INTERFACE I_Logger EXTENDS I_Object

METHOD PUBLIC M_Log
VAR_INPUT
	{attribute 'analysis' := '-33'}
	stEvent	: ST_Event;
END_VAR
END_METHOD

METHOD PUBLIC M_Reset
VAR_INPUT
END_VAR
END_METHOD

END_INTERFACE

(* stored: Version 1.1.0.1
   Itf I_Logger: Id {88be7450-bc52-061e-2cb9-3df6d391e125}
   Method M_Log: Id {6a062c36-2ed5-0ed3-3cfa-49f3c3949c89}
   Method M_Reset: Id {c124a1ce-b4a2-0172-1abe-6ef072f86b26} *)
